TYPE ST_MCRequestChangeMode :
STRUCT

END_STRUCT
END_TYPE

(* stored: Version 1.1.0.1
   DUT ST_MCRequestChangeMode: Id {9bde77f9-3c33-0c5b-34cc-a5aa77e240a2} *)
